FUNCTION_BLOCK FB_TemperatureSensor
VAR_INPUT
END_VAR
VAR_OUTPUT
END_VAR
VAR
	rTemperature : REAL;
	rCorrespondenceFactor : REAL := 0.01;
END_VAR

rTemperature := INT_TO_REAL(MyGVL.iInput1) * rCorrespondenceFactor;

PROPERTY getTemperature : REAL
GET
getTemperature := rTemperature;
END_GET
END_PROPERTY

END_FUNCTION_BLOCK

(* stored: Version 1.1.0.1, ProductVersion 3.1.4024.11
   POU FB_TemperatureSensor: Id {6f346c49-8053-4f07-8a66-62825debe819}, SpecialFunc None
   Property getTemperature: Id {49ba6347-cabd-4894-bd6d-9d1e0d858dbd}
   Get Get: Id {333791c2-d511-43d9-bbb5-4e9f336f4662} *)
